FUNCTION_BLOCK CmdSludgeDischarge (* CAT Function Block Type *)
  (* Standard: 61499-2 *)
  (* Version 0.0, 6/7/2026, Schneider Electric, template *)
  PACKAGE SE.Nereda;
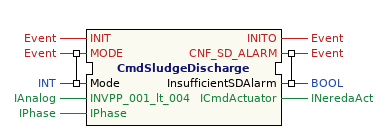
  EVENT_INPUT
    INIT;
    MODE WITH Mode;
  END_EVENT
  EVENT_OUTPUT
    INITO;
    CNF_SD_ALARM WITH InsufficientSDAlarm;
  END_EVENT
  VAR_INPUT
    Mode : INT;
  END_VAR
  VAR_OUTPUT
    InsufficientSDAlarm : BOOL;
  END_VAR
  SOCKETS
    INVPP_001_lt_004 : IAnalog;
    IPhase : IPhase;
  END_SOCKETS
  PLUGS
    ICmdActuator : INeredaAct;
  END_PLUGS
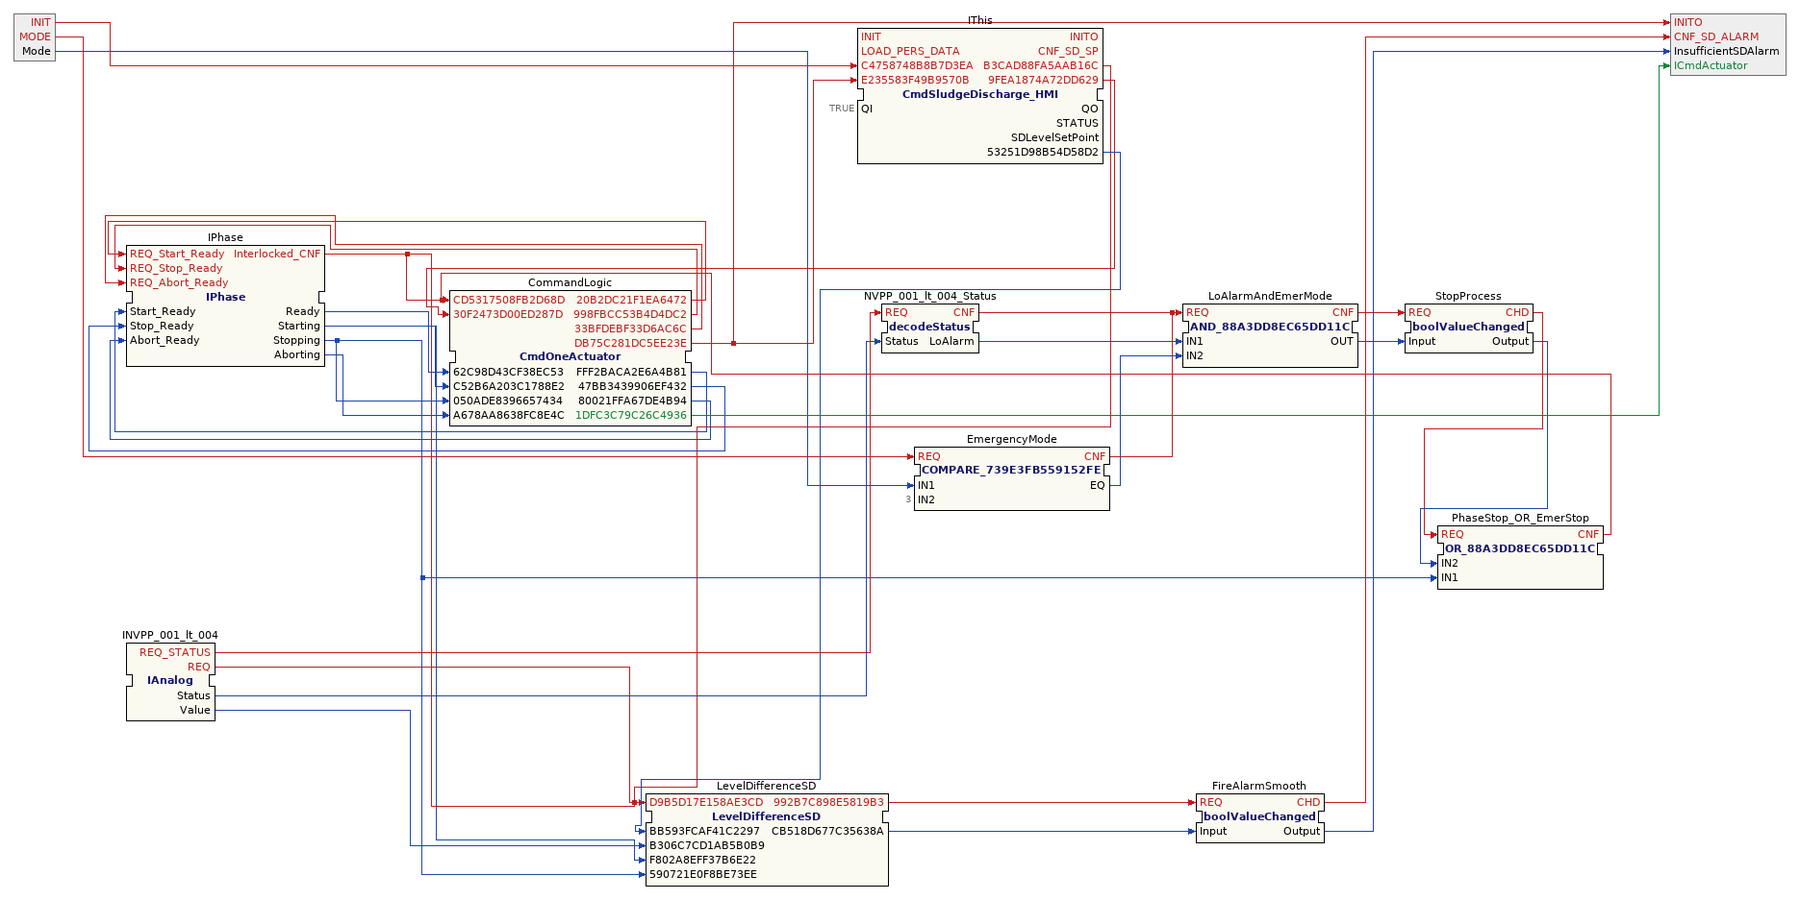
  (* 01 - FUNCTIONNAL INPUT INTERFACE *)
  (* 00 - INITIALIZATION *)
  (* 05 - LOGIC *)
  (* 06 - HMI INTERFACE *)
  (* 03 - FIELD INTERFACE *)
  (* 02 - FUNCTIONNAL OUTPUT INTERFACE *)
  (* Command Logic *)
  (* LoAlarm : Stop Sludge discharge phase reactor during Emergency mode *)
  (* If the level difference is lower than an adjustable value (During Running State), an alarm is generated *)
  FBS
    IThis : CmdSludgeDischarge_HMI(QI := TRUE);
    CommandLogic : CmdOneActuator; {SET_ATTRIBUTE(Configuration.Component.HideUnusedPorts, )}
    NVPP_001_lt_004_Status : decodeStatus; {SET_ATTRIBUTE(Configuration.Component.HideUnusedPorts, )}
    LoAlarmAndEmerMode : AND_88A3DD8EC65DD11C; {SET_ATTRIBUTE(Configuration.GenericFBType.InterfaceParams, Runtime.Standard#CNT:=2;OUT:BOOL)}
    EmergencyMode : COMPARE_739E3FB559152FE(IN2 := 3); {SET_ATTRIBUTE(Configuration.GenericFBType.InterfaceParams, Runtime.Standard#CNT:=2;IN${CNT$}:INT)}
    StopProcess : boolValueChanged;
    PhaseStop_OR_EmerStop : OR_88A3DD8EC65DD11C; {SET_ATTRIBUTE(Configuration.GenericFBType.InterfaceParams, Runtime.Standard#CNT:=2;OUT:BOOL)}
    FireAlarmSmooth : boolValueChanged;
    LevelDifferenceSD : LevelDifferenceSD;
  END_FBS
  EVENT_CONNECTIONS
    INVPP_001_lt_004.REQ_STATUS TO NVPP_001_lt_004_Status.REQ;
    NVPP_001_lt_004_Status.CNF TO LoAlarmAndEmerMode.REQ;
    MODE TO EmergencyMode.REQ;
    EmergencyMode.CNF TO LoAlarmAndEmerMode.REQ;
    LoAlarmAndEmerMode.CNF TO StopProcess.REQ;
    StopProcess.CHD TO PhaseStop_OR_EmerStop.REQ;
    INIT TO IThis.C4758748B8B7D3EA;
    IThis.B3CAD88FA5AAB16C TO LevelDifferenceSD.D9B5D17E158AE3CD;
    INVPP_001_lt_004.REQ TO LevelDifferenceSD.D9B5D17E158AE3CD;
    FireAlarmSmooth.CHD TO CNF_SD_ALARM;
    IPhase.Interlocked_CNF TO CommandLogic.CD5317508FB2D68D;
    IThis.9FEA1874A72DD629 TO CommandLogic.30F2473D00ED287D;
    CommandLogic.20B2DC21F1EA6472 TO IPhase.REQ_Start_Ready;
    CommandLogic.998FBCC53B4D4DC2 TO IPhase.REQ_Stop_Ready;
    CommandLogic.33BFDEBF33D6AC6C TO IPhase.REQ_Abort_Ready;
    CommandLogic.DB75C281DC5EE23E TO INITO;
    CommandLogic.DB75C281DC5EE23E TO IThis.E235583F49B9570B;
    PhaseStop_OR_EmerStop.CNF TO CommandLogic.CD5317508FB2D68D;
    IPhase.Interlocked_CNF TO LevelDifferenceSD.D9B5D17E158AE3CD;
    LevelDifferenceSD.992B7C898E5819B3 TO FireAlarmSmooth.REQ;
  END_CONNECTIONS
  DATA_CONNECTIONS
    INVPP_001_lt_004.Status TO NVPP_001_lt_004_Status.Status;
    NVPP_001_lt_004_Status.LoAlarm TO LoAlarmAndEmerMode.IN1;
    Mode TO EmergencyMode.IN1;
    EmergencyMode.EQ TO LoAlarmAndEmerMode.IN2;
    StopProcess.Output TO PhaseStop_OR_EmerStop.IN2;
    LoAlarmAndEmerMode.OUT TO StopProcess.Input;
    IThis.53251D98B54D58D2 TO LevelDifferenceSD.BB593FCAF41C2297;
    INVPP_001_lt_004.Value TO LevelDifferenceSD.B306C7CD1AB5B0B9;
    FireAlarmSmooth.Output TO InsufficientSDAlarm;
    IPhase.Ready TO CommandLogic.62C98D43CF38EC53;
    IPhase.Starting TO CommandLogic.C52B6A203C1788E2;
    IPhase.Stopping TO CommandLogic.050ADE8396657434;
    IPhase.Aborting TO CommandLogic.A678AA8638FC8E4C;
    CommandLogic.FFF2BACA2E6A4B81 TO IPhase.Start_Ready;
    CommandLogic.47BB3439906EF432 TO IPhase.Stop_Ready;
    CommandLogic.80021FFA67DE4B94 TO IPhase.Abort_Ready;
    IPhase.Stopping TO PhaseStop_OR_EmerStop.IN1;
    LevelDifferenceSD.CB518D677C35638A TO FireAlarmSmooth.Input;
    IPhase.Starting TO LevelDifferenceSD.F802A8EFF37B6E22;
    IPhase.Stopping TO LevelDifferenceSD.590721E0F8BE73EE;
  END_CONNECTIONS
  ADAPTER_CONNECTIONS
    CommandLogic.1DFC3C79C26C4936 TO ICmdActuator;
  END_CONNECTIONS
END_FUNCTION_BLOCK
